// Mitsubishi GX Works2 project: 0206 서보 2축   PLC: Q03UDV

PROGRAM MAIN
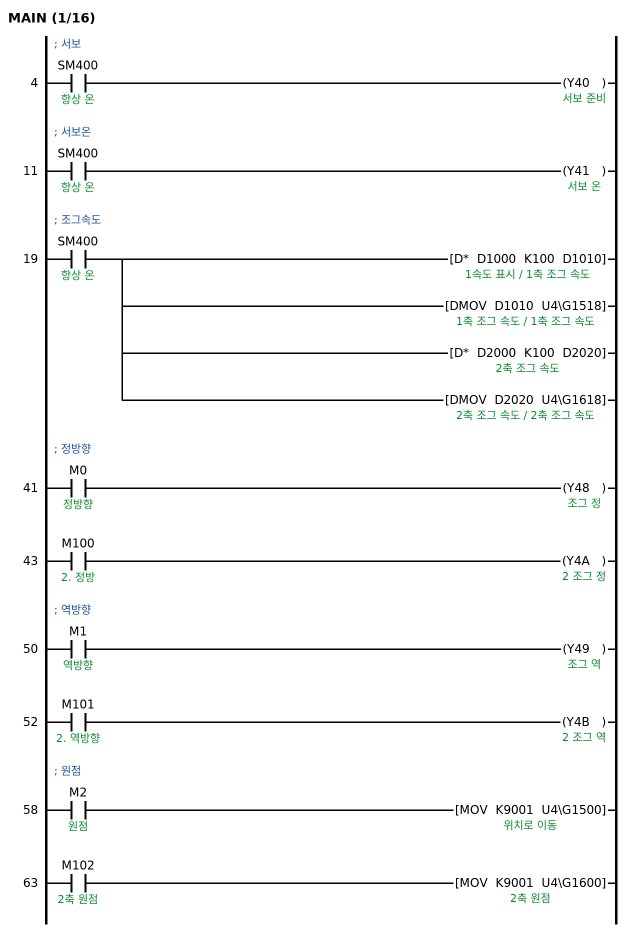
; 서보
4     LD      SM400  ; 항상 온
      OUT     Y40  ; 서보 준비
; 서보온
11    LD      SM400  ; 항상 온
      OUT     Y41  ; 서보 온
; 조그속도
19    LD      SM400  ; 항상 온
      D*      D1000 K100 D1010  ; 1속도 표시 / 1축 조그 속도
      DMOV    D1010 U4\G1518  ; 1축 조그 속도
      D*      D2000 K100 D2020  ; 2축 조그 속도
      DMOV    D2020 U4\G1618  ; 2축 조그 속도
; 정방향
41    LD      M0  ; 정방향
      OUT     Y48  ; 조그 정
43    LD      M100  ; 2. 정방
      OUT     Y4A  ; 2 조그 정
; 역방향
50    LD      M1  ; 역방향
      OUT     Y49  ; 조그 역
52    LD      M101  ; 2. 역방향
      OUT     Y4B  ; 2 조그 역
; 원점
58    LD      M2  ; 원점
      MOV     K9001 U4\G1500  ; 위치로 이동
63    LD      M102  ; 2축 원점
      MOV     K9001 U4\G1600  ; 2축 원점
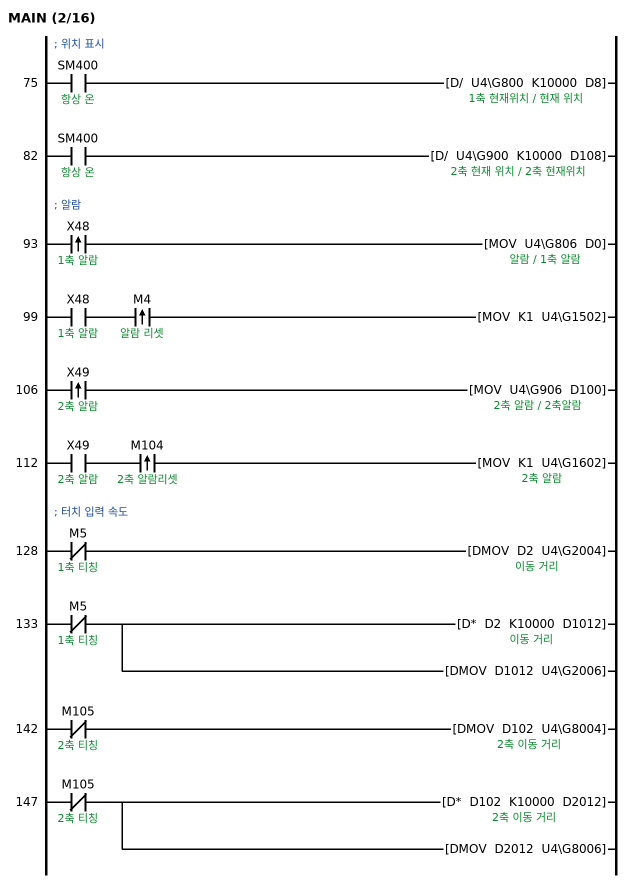
; 위치 표시
75    LD      SM400  ; 항상 온
      D/      U4\G800 K10000 D8  ; 1축 현재위치 / 현재 위치
82    LD      SM400  ; 항상 온
      D/      U4\G900 K10000 D108  ; 2축 현재 위치 / 2축 현재위치
; 알람
93    LDP     X48  ; 1축 알람
      MOV     U4\G806 D0  ; 알람 / 1축 알람
99    LD      X48  ; 1축 알람
      ANDP    M4  ; 알람 리셋
      MOV     K1 U4\G1502
106   LDP     X49  ; 2축 알람
      MOV     U4\G906 D100  ; 2축 알람 / 2축알람
112   LD      X49  ; 2축 알람
      ANDP    M104  ; 2축 알람리셋
      MOV     K1 U4\G1602  ; 2축 알람
; 터치 입력 속도
128   LDI     M5  ; 1축 티칭
      DMOV    D2 U4\G2004  ; 이동 거리
133   LDI     M5  ; 1축 티칭
      D*      D2 K10000 D1012
      DMOV    D1012 U4\G2006
142   LDI     M105  ; 2축 티칭
      DMOV    D102 U4\G8004  ; 2축 이동 거리
147   LDI     M105  ; 2축 티칭
      D*      D102 K10000 D2012
      DMOV    D2012 U4\G8006
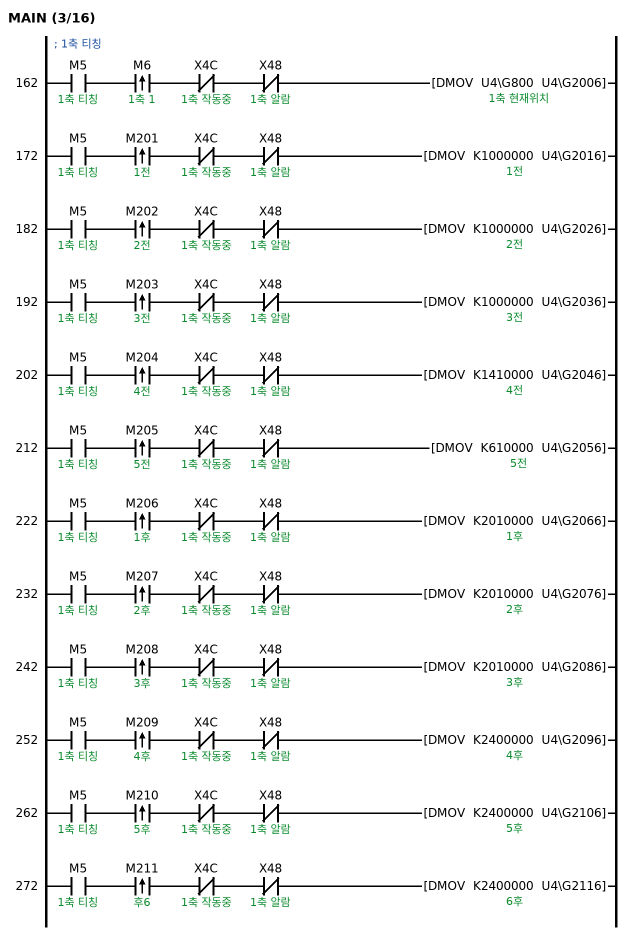
; 1축 티칭
162   LD      M5  ; 1축 티칭
      ANDP    M6  ; 1축 1
      ANI     X4C  ; 1축 작동중
      ANI     X48  ; 1축 알람
      DMOV    U4\G800 U4\G2006
172   LD      M5  ; 1축 티칭
      ANDP    M201  ; 1전
      ANI     X4C  ; 1축 작동중
      ANI     X48  ; 1축 알람
      DMOV    K1000000 U4\G2016  ; 1전
182   LD      M5  ; 1축 티칭
      ANDP    M202  ; 2전
      ANI     X4C  ; 1축 작동중
      ANI     X48  ; 1축 알람
      DMOV    K1000000 U4\G2026  ; 2전
192   LD      M5  ; 1축 티칭
      ANDP    M203  ; 3전
      ANI     X4C  ; 1축 작동중
      ANI     X48  ; 1축 알람
      DMOV    K1000000 U4\G2036  ; 3전
202   LD      M5  ; 1축 티칭
      ANDP    M204  ; 4전
      ANI     X4C  ; 1축 작동중
      ANI     X48  ; 1축 알람
      DMOV    K1410000 U4\G2046  ; 4전
212   LD      M5  ; 1축 티칭
      ANDP    M205  ; 5전
      ANI     X4C  ; 1축 작동중
      ANI     X48  ; 1축 알람
      DMOV    K610000 U4\G2056  ; 5전
222   LD      M5  ; 1축 티칭
      ANDP    M206  ; 1후
      ANI     X4C  ; 1축 작동중
      ANI     X48  ; 1축 알람
      DMOV    K2010000 U4\G2066  ; 1후
232   LD      M5  ; 1축 티칭
      ANDP    M207  ; 2후
      ANI     X4C  ; 1축 작동중
      ANI     X48  ; 1축 알람
      DMOV    K2010000 U4\G2076  ; 2후
242   LD      M5  ; 1축 티칭
      ANDP    M208  ; 3후
      ANI     X4C  ; 1축 작동중
      ANI     X48  ; 1축 알람
      DMOV    K2010000 U4\G2086  ; 3후
252   LD      M5  ; 1축 티칭
      ANDP    M209  ; 4후
      ANI     X4C  ; 1축 작동중
      ANI     X48  ; 1축 알람
      DMOV    K2400000 U4\G2096  ; 4후
262   LD      M5  ; 1축 티칭
      ANDP    M210  ; 5후
      ANI     X4C  ; 1축 작동중
      ANI     X48  ; 1축 알람
      DMOV    K2400000 U4\G2106  ; 5후
272   LD      M5  ; 1축 티칭
      ANDP    M211  ; 후6
      ANI     X4C  ; 1축 작동중
      ANI     X48  ; 1축 알람
      DMOV    K2400000 U4\G2116  ; 6후
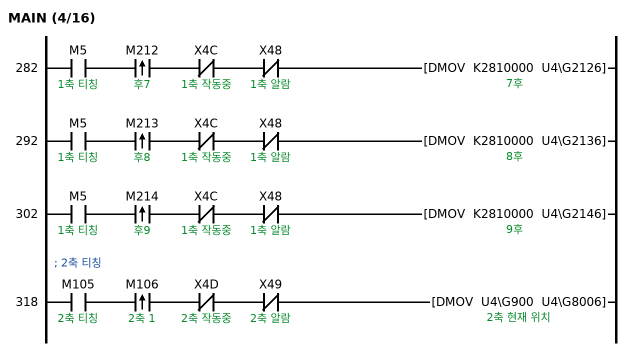
282   LD      M5  ; 1축 티칭
      ANDP    M212  ; 후7
      ANI     X4C  ; 1축 작동중
      ANI     X48  ; 1축 알람
      DMOV    K2810000 U4\G2126  ; 7후
292   LD      M5  ; 1축 티칭
      ANDP    M213  ; 후8
      ANI     X4C  ; 1축 작동중
      ANI     X48  ; 1축 알람
      DMOV    K2810000 U4\G2136  ; 8후
302   LD      M5  ; 1축 티칭
      ANDP    M214  ; 후9
      ANI     X4C  ; 1축 작동중
      ANI     X48  ; 1축 알람
      DMOV    K2810000 U4\G2146  ; 9후
; 2축 티칭
318   LD      M105  ; 2축 티칭
      ANDP    M106  ; 2축 1
      ANI     X4D  ; 2축 작동중
      ANI     X49  ; 2축 알람
      DMOV    U4\G900 U4\G8006
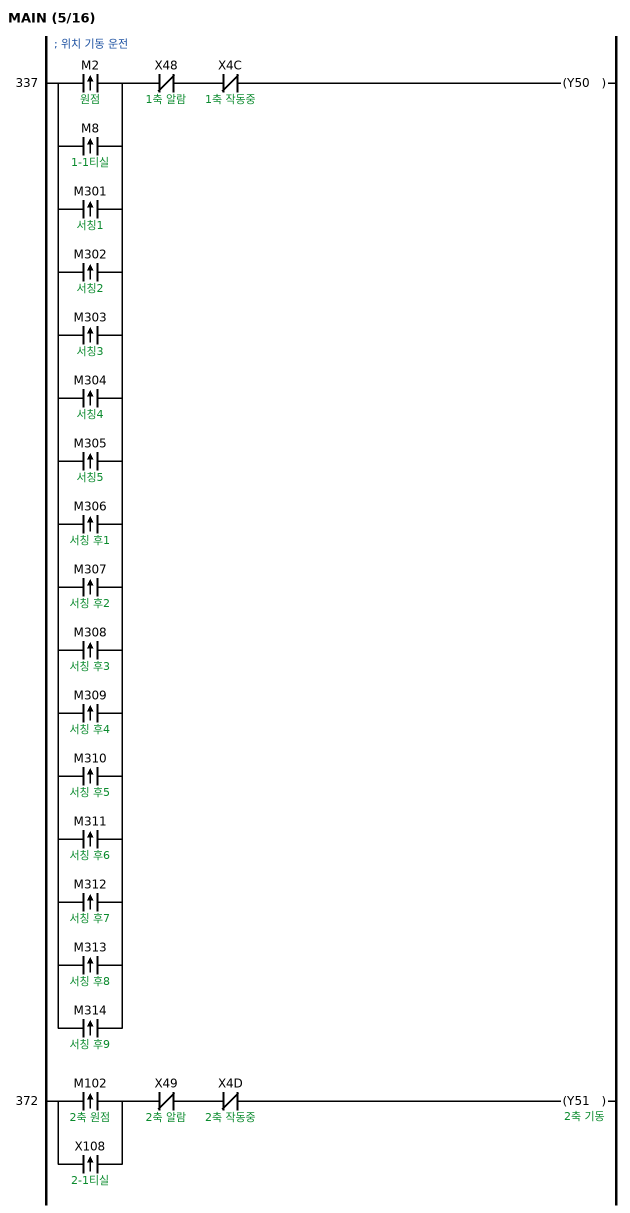
; 위치 기동 운전
337   LDP     M2  ; 원점
      ORP     M8  ; 1-1티실
      ORP     M301  ; 서칭1
      ORP     M302  ; 서칭2
      ORP     M303  ; 서칭3
      ORP     M304  ; 서칭4
      ORP     M305  ; 서칭5
      ORP     M306  ; 서칭 후1
      ORP     M307  ; 서칭 후2
      ORP     M308  ; 서칭 후3
      ORP     M309  ; 서칭 후4
      ORP     M310  ; 서칭 후5
      ORP     M311  ; 서칭 후6
      ORP     M312  ; 서칭 후7
      ORP     M313  ; 서칭 후8
      ORP     M314  ; 서칭 후9
      ANI     X48  ; 1축 알람
      ANI     X4C  ; 1축 작동중
      OUT     Y50
372   LDP     M102  ; 2축 원점
      ORP     X108  ; 2-1티실
      ANI     X49  ; 2축 알람
      ANI     X4D  ; 2축 작동중
      OUT     Y51  ; 2축 기동
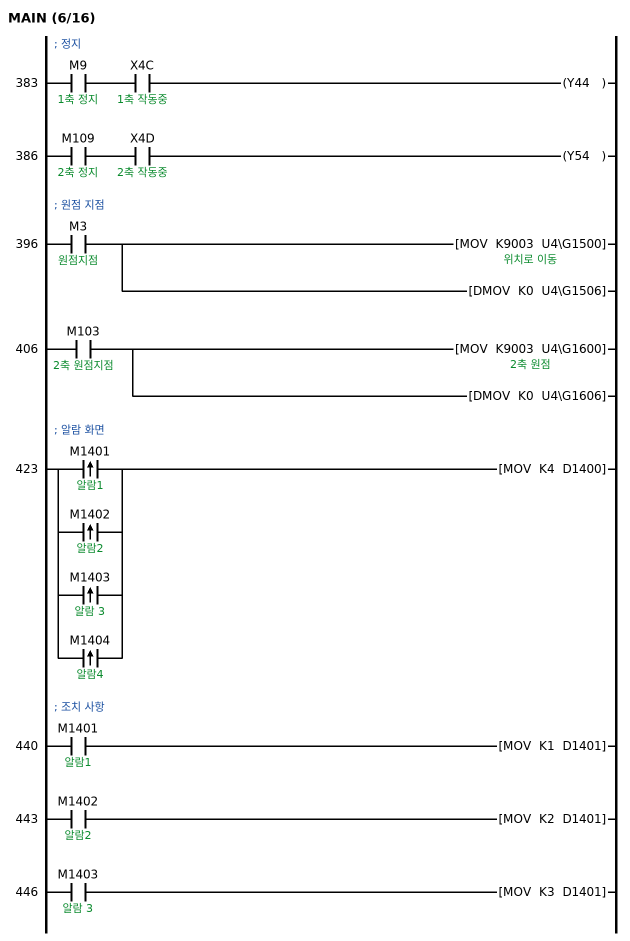
; 정지
383   LD      M9  ; 1축 정지
      AND     X4C  ; 1축 작동중
      OUT     Y44
386   LD      M109  ; 2축 정지
      AND     X4D  ; 2축 작동중
      OUT     Y54
; 원점 지점
396   LD      M3  ; 원점지점
      MOV     K9003 U4\G1500
      DMOV    K0 U4\G1506
406   LD      M103  ; 2축 원점지점
      MOV     K9003 U4\G1600
      DMOV    K0 U4\G1606
; 알람 화면
423   LDP     M1401  ; 알람1
      ORP     M1402  ; 알람2
      ORP     M1403  ; 알람 3
      ORP     M1404  ; 알람4
      MOV     K4 D1400
; 조치 사항
440   LD      M1401  ; 알람1
      MOV     K1 D1401
443   LD      M1402  ; 알람2
      MOV     K2 D1401
446   LD      M1403  ; 알람 3
      MOV     K3 D1401
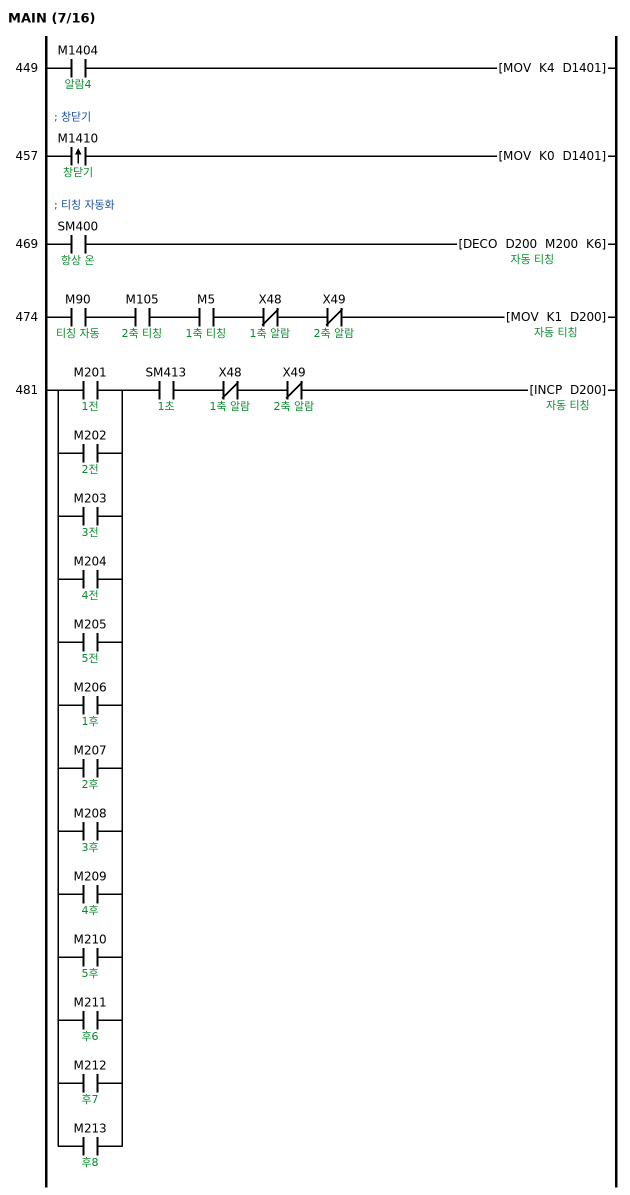
449   LD      M1404  ; 알람4
      MOV     K4 D1401
; 창닫기
457   LDP     M1410  ; 창닫기
      MOV     K0 D1401
; 티칭 자동화
469   LD      SM400  ; 항상 온
      DECO    D200 M200 K6  ; 자동 티칭
474   LD      M90  ; 티칭 자동
      AND     M105  ; 2축 티칭
      AND     M5  ; 1축 티칭
      ANI     X48  ; 1축 알람
      ANI     X49  ; 2축 알람
      MOV     K1 D200
481   LD      M201  ; 1전
      OR      M202  ; 2전
      OR      M203  ; 3전
      OR      M204  ; 4전
      OR      M205  ; 5전
      OR      M206  ; 1후
      OR      M207  ; 2후
      OR      M208  ; 3후
      OR      M209  ; 4후
      OR      M210  ; 5후
      OR      M211  ; 후6
      OR      M212  ; 후7
      OR      M213  ; 후8
      AND     SM413  ; 1초
      ANI     X48  ; 1축 알람
      ANI     X49  ; 2축 알람
      INCP    D200
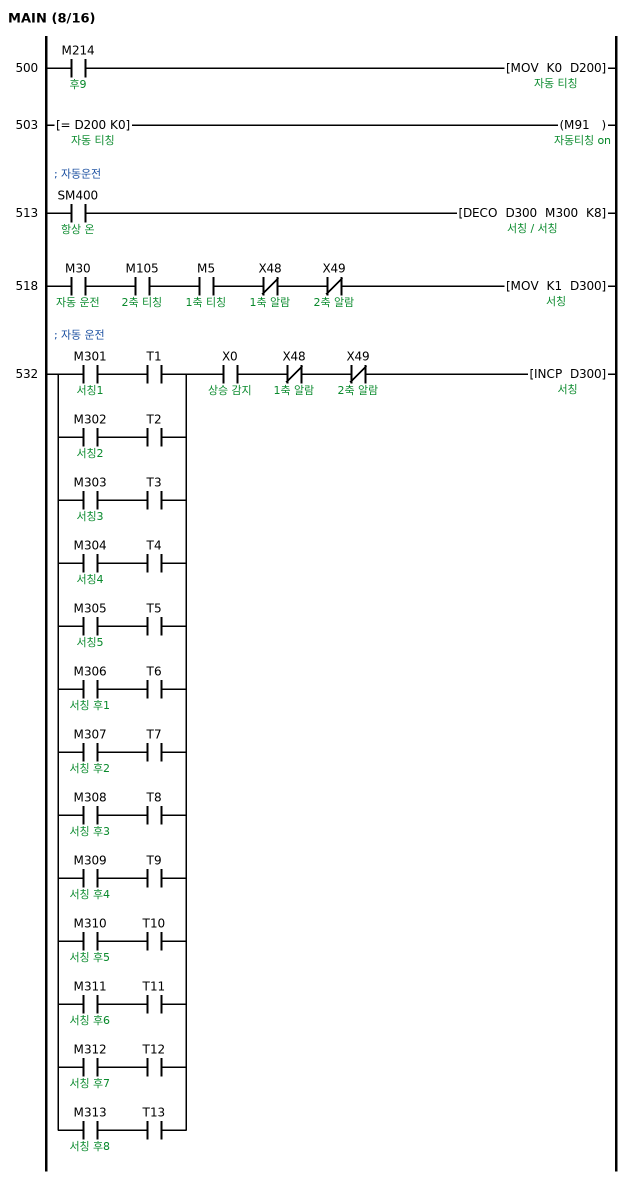
500   LD      M214  ; 후9
      MOV     K0 D200
503   LD=     D200 K0  ; 자동 티칭
      OUT     M91  ; 자동티칭 on
; 자동운전
513   LD      SM400  ; 항상 온
      DECO    D300 M300 K8  ; 서칭 / 서칭
518   LD      M30  ; 자동 운전
      AND     M105  ; 2축 티칭
      AND     M5  ; 1축 티칭
      ANI     X48  ; 1축 알람
      ANI     X49  ; 2축 알람
      MOV     K1 D300
; 자동 운전
532   LD      M301  ; 서칭1
      AND     T1
      LD      M302  ; 서칭2
      AND     T2
      ORB
      LD      M303  ; 서칭3
      AND     T3
      ORB
      LD      M304  ; 서칭4
      AND     T4
      ORB
      LD      M305  ; 서칭5
      AND     T5
      ORB
      LD      M306  ; 서칭 후1
      AND     T6
      ORB
      LD      M307  ; 서칭 후2
      AND     T7
      ORB
      LD      M308  ; 서칭 후3
      AND     T8
      ORB
      LD      M309  ; 서칭 후4
      AND     T9
      ORB
      LD      M310  ; 서칭 후5
      AND     T10
      ORB
      LD      M311  ; 서칭 후6
      AND     T11
      ORB
      LD      M312  ; 서칭 후7
      AND     T12
      ORB
      LD      M313  ; 서칭 후8
      AND     T13
      ORB
      AND     X0  ; 상승 감지
      ANI     X48  ; 1축 알람
      ANI     X49  ; 2축 알람
      INCP    D300
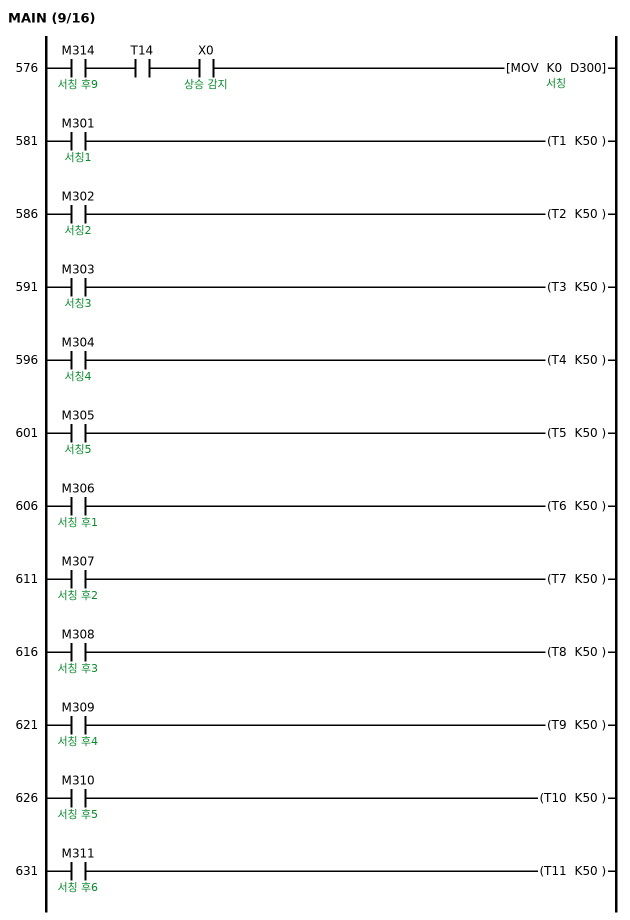
576   LD      M314  ; 서칭 후9
      AND     T14
      AND     X0  ; 상승 감지
      MOV     K0 D300
581   LD      M301  ; 서칭1
      OUT     T1 K50
586   LD      M302  ; 서칭2
      OUT     T2 K50
591   LD      M303  ; 서칭3
      OUT     T3 K50
596   LD      M304  ; 서칭4
      OUT     T4 K50
601   LD      M305  ; 서칭5
      OUT     T5 K50
606   LD      M306  ; 서칭 후1
      OUT     T6 K50
611   LD      M307  ; 서칭 후2
      OUT     T7 K50
616   LD      M308  ; 서칭 후3
      OUT     T8 K50
621   LD      M309  ; 서칭 후4
      OUT     T9 K50
626   LD      M310  ; 서칭 후5
      OUT     T10 K50
631   LD      M311  ; 서칭 후6
      OUT     T11 K50
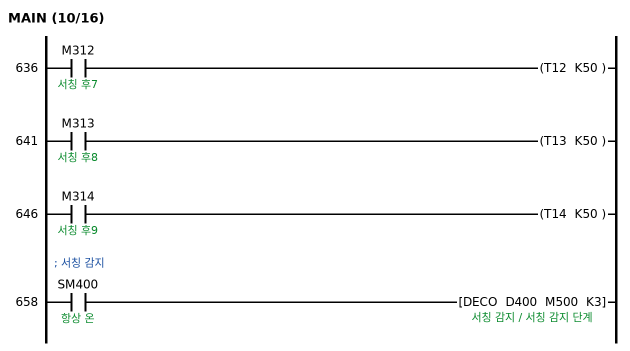
636   LD      M312  ; 서칭 후7
      OUT     T12 K50
641   LD      M313  ; 서칭 후8
      OUT     T13 K50
646   LD      M314  ; 서칭 후9
      OUT     T14 K50
; 서칭 감지
658   LD      SM400  ; 항상 온
      DECO    D400 M500 K3  ; 서칭 감지 / 서칭 감지 단계
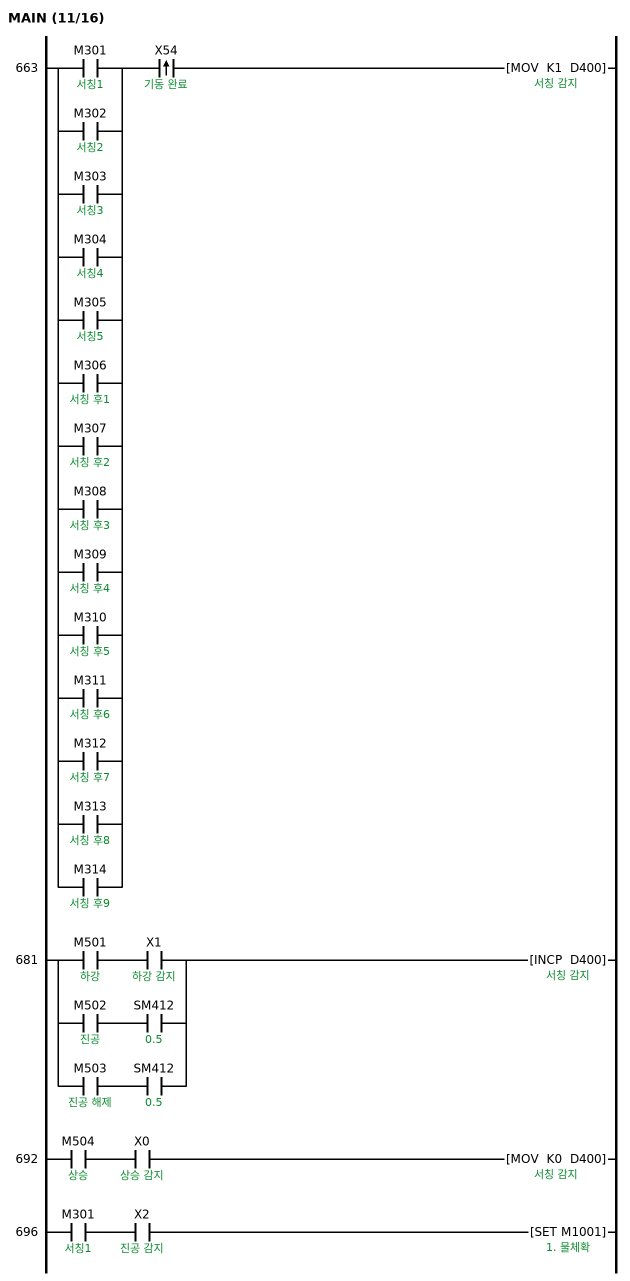
663   LD      M301  ; 서칭1
      OR      M302  ; 서칭2
      OR      M303  ; 서칭3
      OR      M304  ; 서칭4
      OR      M305  ; 서칭5
      OR      M306  ; 서칭 후1
      OR      M307  ; 서칭 후2
      OR      M308  ; 서칭 후3
      OR      M309  ; 서칭 후4
      OR      M310  ; 서칭 후5
      OR      M311  ; 서칭 후6
      OR      M312  ; 서칭 후7
      OR      M313  ; 서칭 후8
      OR      M314  ; 서칭 후9
      ANDP    X54  ; 기동 완료
      MOV     K1 D400
681   LD      M501  ; 하강
      AND     X1  ; 하강 감지
      LD      M502  ; 진공
      AND     SM412  ; 0.5
      ORB
      LD      M503  ; 진공 해제
      AND     SM412  ; 0.5
      ORB
      INCP    D400
692   LD      M504  ; 상승
      AND     X0  ; 상승 감지
      MOV     K0 D400
696   LD      M301  ; 서칭1
      AND     X2  ; 진공 감지
      SET     M1001  ; 1. 물체확
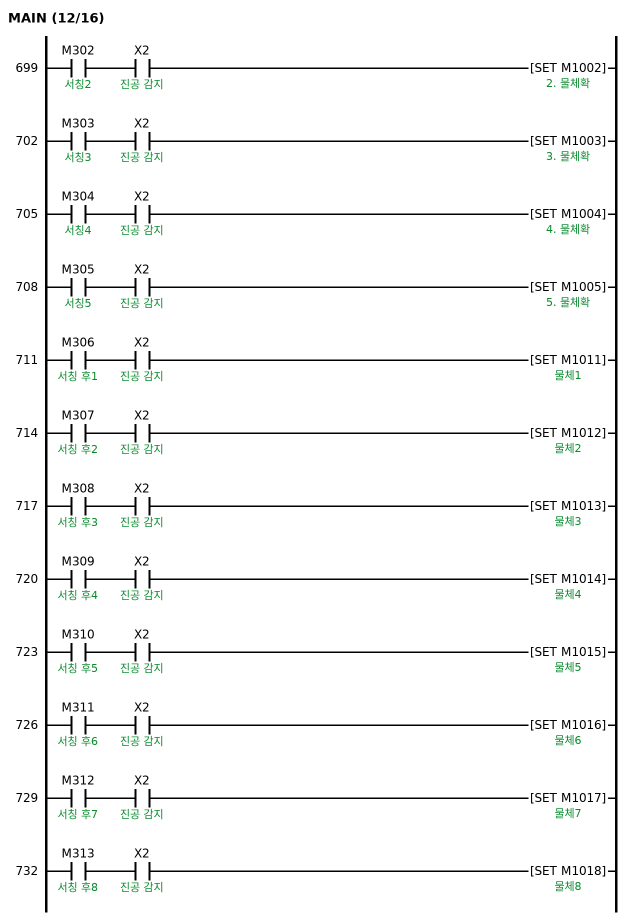
699   LD      M302  ; 서칭2
      AND     X2  ; 진공 감지
      SET     M1002  ; 2. 물체확
702   LD      M303  ; 서칭3
      AND     X2  ; 진공 감지
      SET     M1003  ; 3. 물체확
705   LD      M304  ; 서칭4
      AND     X2  ; 진공 감지
      SET     M1004  ; 4. 물체확
708   LD      M305  ; 서칭5
      AND     X2  ; 진공 감지
      SET     M1005  ; 5. 물체확
711   LD      M306  ; 서칭 후1
      AND     X2  ; 진공 감지
      SET     M1011  ; 물체1
714   LD      M307  ; 서칭 후2
      AND     X2  ; 진공 감지
      SET     M1012  ; 물체2
717   LD      M308  ; 서칭 후3
      AND     X2  ; 진공 감지
      SET     M1013  ; 물체3
720   LD      M309  ; 서칭 후4
      AND     X2  ; 진공 감지
      SET     M1014  ; 물체4
723   LD      M310  ; 서칭 후5
      AND     X2  ; 진공 감지
      SET     M1015  ; 물체5
726   LD      M311  ; 서칭 후6
      AND     X2  ; 진공 감지
      SET     M1016  ; 물체6
729   LD      M312  ; 서칭 후7
      AND     X2  ; 진공 감지
      SET     M1017  ; 물체7
732   LD      M313  ; 서칭 후8
      AND     X2  ; 진공 감지
      SET     M1018  ; 물체8
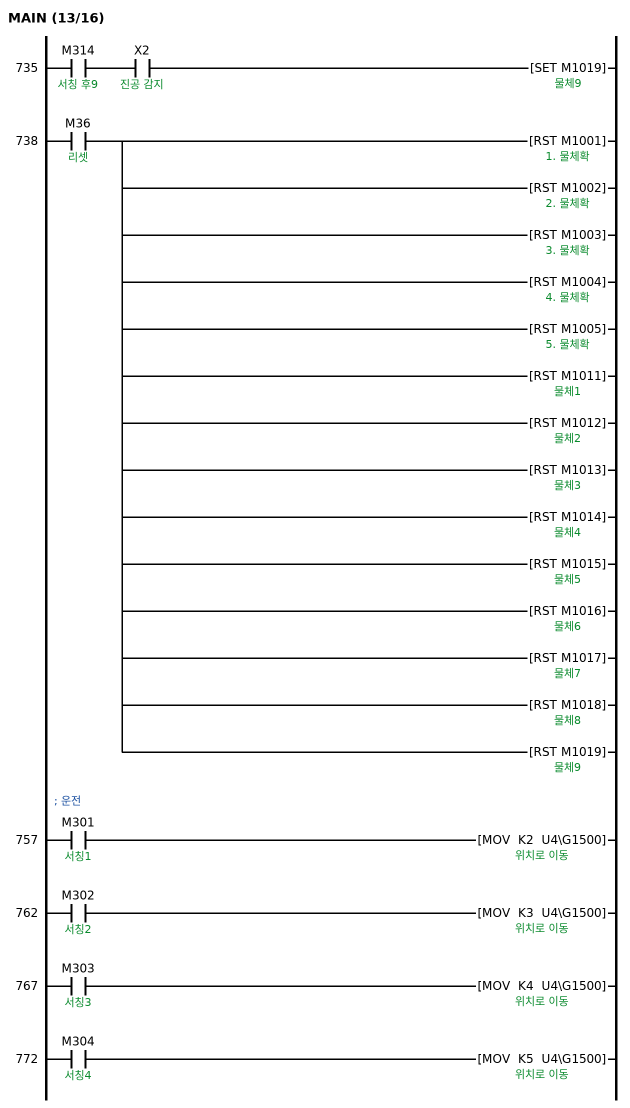
735   LD      M314  ; 서칭 후9
      AND     X2  ; 진공 감지
      SET     M1019  ; 물체9
738   LD      M36  ; 리셋
      RST     M1001  ; 1. 물체확
      RST     M1002  ; 2. 물체확
      RST     M1003  ; 3. 물체확
      RST     M1004  ; 4. 물체확
      RST     M1005  ; 5. 물체확
      RST     M1011  ; 물체1
      RST     M1012  ; 물체2
      RST     M1013  ; 물체3
      RST     M1014  ; 물체4
      RST     M1015  ; 물체5
      RST     M1016  ; 물체6
      RST     M1017  ; 물체7
      RST     M1018  ; 물체8
      RST     M1019  ; 물체9
; 운전
757   LD      M301  ; 서칭1
      MOV     K2 U4\G1500
762   LD      M302  ; 서칭2
      MOV     K3 U4\G1500
767   LD      M303  ; 서칭3
      MOV     K4 U4\G1500
772   LD      M304  ; 서칭4
      MOV     K5 U4\G1500
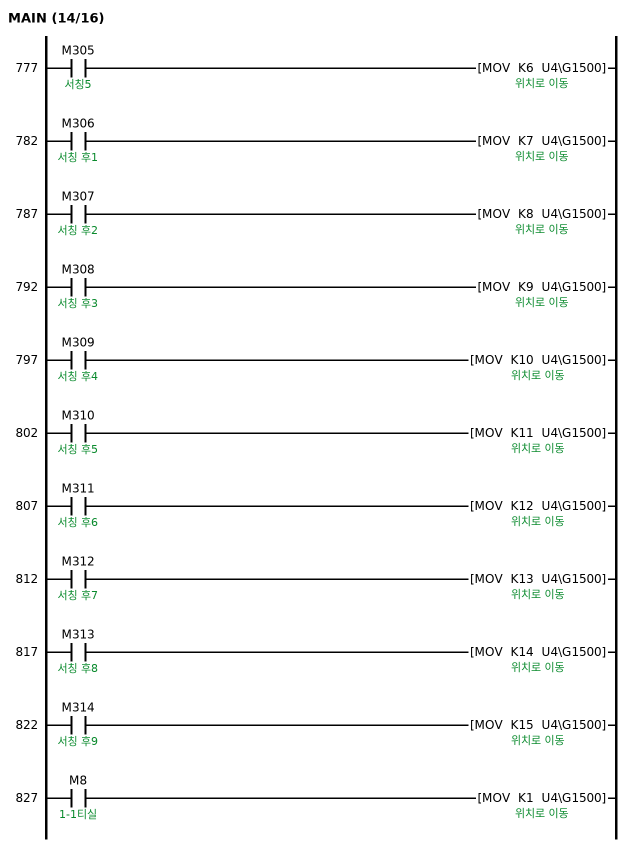
777   LD      M305  ; 서칭5
      MOV     K6 U4\G1500
782   LD      M306  ; 서칭 후1
      MOV     K7 U4\G1500
787   LD      M307  ; 서칭 후2
      MOV     K8 U4\G1500
792   LD      M308  ; 서칭 후3
      MOV     K9 U4\G1500
797   LD      M309  ; 서칭 후4
      MOV     K10 U4\G1500
802   LD      M310  ; 서칭 후5
      MOV     K11 U4\G1500
807   LD      M311  ; 서칭 후6
      MOV     K12 U4\G1500
812   LD      M312  ; 서칭 후7
      MOV     K13 U4\G1500
817   LD      M313  ; 서칭 후8
      MOV     K14 U4\G1500
822   LD      M314  ; 서칭 후9
      MOV     K15 U4\G1500
827   LD      M8  ; 1-1티실
      MOV     K1 U4\G1500
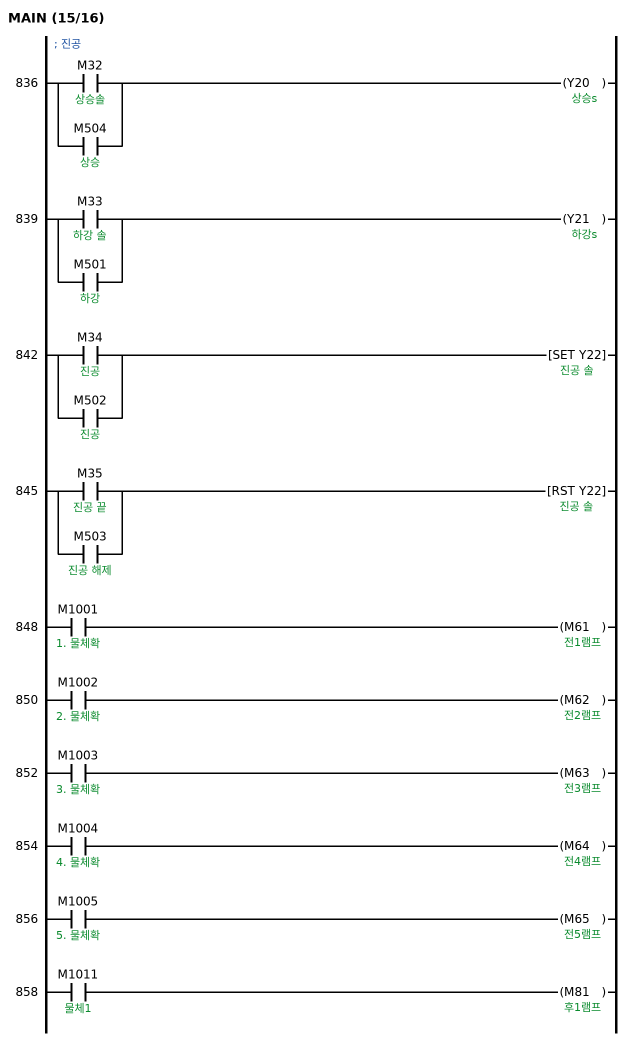
; 진공
836   LD      M32  ; 상승솔
      OR      M504  ; 상승
      OUT     Y20  ; 상승s
839   LD      M33  ; 하강 솔
      OR      M501  ; 하강
      OUT     Y21  ; 하강s
842   LD      M34  ; 진공
      OR      M502  ; 진공
      SET     Y22  ; 진공 솔
845   LD      M35  ; 진공 끝
      OR      M503  ; 진공 해제
      RST     Y22  ; 진공 솔
848   LD      M1001  ; 1. 물체확
      OUT     M61  ; 전1램프
850   LD      M1002  ; 2. 물체확
      OUT     M62  ; 전2램프
852   LD      M1003  ; 3. 물체확
      OUT     M63  ; 전3램프
854   LD      M1004  ; 4. 물체확
      OUT     M64  ; 전4램프
856   LD      M1005  ; 5. 물체확
      OUT     M65  ; 전5램프
858   LD      M1011  ; 물체1
      OUT     M81  ; 후1램프
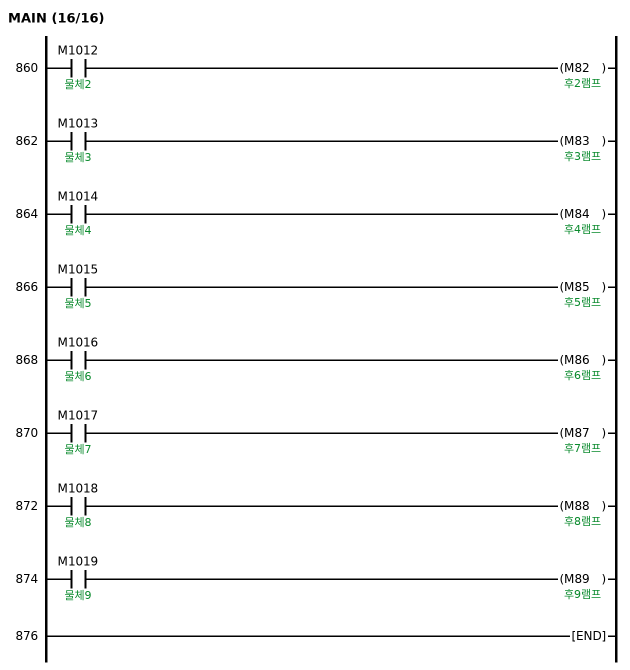
860   LD      M1012  ; 물체2
      OUT     M82  ; 후2램프
862   LD      M1013  ; 물체3
      OUT     M83  ; 후3램프
864   LD      M1014  ; 물체4
      OUT     M84  ; 후4램프
866   LD      M1015  ; 물체5
      OUT     M85  ; 후5램프
868   LD      M1016  ; 물체6
      OUT     M86  ; 후6램프
870   LD      M1017  ; 물체7
      OUT     M87  ; 후7램프
872   LD      M1018  ; 물체8
      OUT     M88  ; 후8램프
874   LD      M1019  ; 물체9
      OUT     M89  ; 후9램프
876   END
END_PROGRAM

// device comments not shown above
M7  ; 1축 2
M107  ; 2축 2
M400  ; 서칭 감지단계
M401  ; 알람 1
M402  ; 알람2
M403  ; 알람 3
M404  ; 알람 4
M410  ; 창 닫기
M1022  ; 물체2
D101  ; 소수점제
